{attribute 'GeneratedUsingTerminal: EL2911-0000-0016'}
{attribute addProperty BoxType "EL2911-0000-0016"}
{attribute addProperty Id "Standard_OutputAT %Q*BOOL1"}
{attribute addProperty CRC "2731189318"}
{attribute addProperty Size "1"}
TYPE Outputs_A2CAA446 :
STRUCT
	{attribute addProperty Name "Standard_Output"}
	Standard_Output AT %Q* : BOOL;
END_STRUCT
END_TYPE

(* stored: Version 1.2.0.0, ProductVersion 3.1.4024.9
   DUT Outputs_A2CAA446: Id {7f2e91c7-fab7-4014-beab-a10debf1afff} *)
